{attribute 'qualified_only'}
{attribute 'strict'}
{attribute 'to_string'}
TYPE ST130_Cylinders_e :
(
    Kammer_Offnen_Links,
    Kammer_Offnen_Rechts,
    Kammer_nachfullen_Links,
    Kammer_nachfullen_Rechts,
    Vibrieren_Kammer_Links,
    Vibrieren_Kammer_Rechts,
    Niederhalter_Patrone,
    Vibrienren_Patrone_Links,
    Viebrieren_Patrone_Rechts
);
END_TYPE

(* stored: Version 1.1.0.1, ProductVersion 3.1.4024.6
   EnumerationTextList ST130_Cylinders_e: Id {ff7bf38d-e7fd-4f27-9d60-c41db9f00c2d} *)
